// TIA Portal V17 export
// export: Created 2022-03-12T16:05:34.4615389Z, ExportSetting WithDefaults, DisplayName Totally Integrated Automation Portal, DisplayVersion V17, DisplayName TIA Portal Openness, DisplayVersion V17, DisplayName TIA Portal Version Control Interface, DisplayVersion V17, DisplayName STEP 7 Professional, DisplayVersion V17, DisplayName STEP 7 Safety, DisplayVersion V17, DisplayName WinCC Advanced / Unified PC, DisplayVersion V17
TYPE "CPG_typeEventSummation"
// stored: IsFailsafeCompliant false
   STRUCT
      sts_FirstOutEvent { S7_SetPoint := 'True'} : "CPG_typeEvent";   // First Out (Stop Reason) Event
      sts_FirstOutEventCat { S7_SetPoint := 'True'} : Array[0..9] of "CPG_typeEvent";   // First Out (Stop Reason) Event by Category\
      sts_Events { S7_SetPoint := 'True'} : Array[0.."CPG_NO_OF_STS_ELEMENTS_EVENT_SUM_UPPER_LIM"] of "CPG_typeEvent";   // All Active Events
      sts_NumEvents : Int;   // Number of Active Events
      sts_Category_0_Latched : Bool;   // Category 0 Event - latched (require reset cmd)
      sts_Category_1_Latched : Bool;   // Category 1 Event - latched (require reset cmd)
      sts_Category_2_Latched : Bool;   // Category 2 Event - latched (require reset cmd)
      sts_Category_3_Latched : Bool;   // Category 3 Event - latched (require reset cmd)
      sts_Category_4_Latched : Bool;   // Category 4 Event - latched (require reset cmd)
      sts_Category_5_Latched : Bool;   // Category 5 Event - latched (require reset cmd)
      sts_Category_6_Latched : Bool;   // Category 6 Event - latched (require reset cmd)
      sts_Category_7_Latched : Bool;   // Category 7 Event - latched (require reset cmd)
      sts_Category_8_Latched : Bool;   // Category 8 Event - latched (require reset cmd)
      sts_Category_9_Latched : Bool;   // Category 9 Event - latched (require reset cmd)
      sts_Category_0_NotLatched : Bool;   // Category 0 Event - NotLatched (currently active)
      sts_Category_1_NotLatched : Bool;   // Category 1 Event - NotLatched (currently active)
      sts_Category_2_NotLatched : Bool;   // Category 2 Event - NotLatched (currently active)
      sts_Category_3_NotLatched : Bool;   // Category 3 Event - NotLatched (currently active)
      sts_Category_4_NotLatched : Bool;   // Category 4 Event - NotLatched (currently active)
      sts_Category_5_NotLatched : Bool;   // Category 5 Event - NotLatched (currently active)
      sts_Category_6_NotLatched : Bool;   // Category 6 Event - NotLatched (currently active)
      sts_Category_7_NotLatched : Bool;   // Category 7 Event - NotLatched (currently active)
      sts_Category_8_NotLatched : Bool;   // Category 8 Event - NotLatched (currently active)
      sts_Category_9_NotLatched : Bool;   // Category 9 Event - NotLatched (currently active)
      sts_CurrentActiveEvent : Bool;   // Event Active = 1, not active = 0
      wrk_EventArraySize : Int;   // Maximum Array Size - DO NOT MODIFY
      wrk_Category_0_Latched : Bool;   // Working Variable - DO NOT MODIFY
      wrk_Category_1_Latched : Bool;   // Working Variable - DO NOT MODIFY
      wrk_Category_2_Latched : Bool;   // Working Variable - DO NOT MODIFY
      wrk_Category_3_Latched : Bool;   // Working Variable - DO NOT MODIFY
      wrk_Category_4_Latched : Bool;   // Working Variable - DO NOT MODIFY
      wrk_Category_5_Latched : Bool;   // Working Variable - DO NOT MODIFY
      wrk_Category_6_Latched : Bool;   // Working Variable - DO NOT MODIFY
      wrk_Category_7_Latched : Bool;   // Working Variable - DO NOT MODIFY
      wrk_Category_8_Latched : Bool;   // Working Variable - DO NOT MODIFY
      wrk_Category_9_Latched : Bool;   // Working Variable - DO NOT MODIFY
      wrk_Category_0_NotLatched : Bool;   // Working Variable - DO NOT MODIFY
      wrk_Category_1_NotLatched : Bool;   // Working Variable - DO NOT MODIFY
      wrk_Category_2_NotLatched : Bool;   // Working Variable - DO NOT MODIFY
      wrk_Category_3_NotLatched : Bool;   // Working Variable - DO NOT MODIFY
      wrk_Category_4_NotLatched : Bool;   // Working Variable - DO NOT MODIFY
      wrk_Category_5_NotLatched : Bool;   // Working Variable - DO NOT MODIFY
      wrk_Category_6_NotLatched : Bool;   // Working Variable - DO NOT MODIFY
      wrk_Category_7_NotLatched : Bool;   // Working Variable - DO NOT MODIFY
      wrk_Category_8_NotLatched : Bool;   // Working Variable - DO NOT MODIFY
      wrk_Category_9_NotLatched : Bool;   // Working Variable - DO NOT MODIFY
      wrk_CurrentActiveEvent : Bool;   // Working Variable - DO NOT MODIFY
   END_STRUCT;
END_TYPE
